PROGRAM MotionControl
VAR
END_VAR

SingleAxis_LD();

METHOD SingleAxis_LD : BOOL
VAR_INPUT
END_VAR
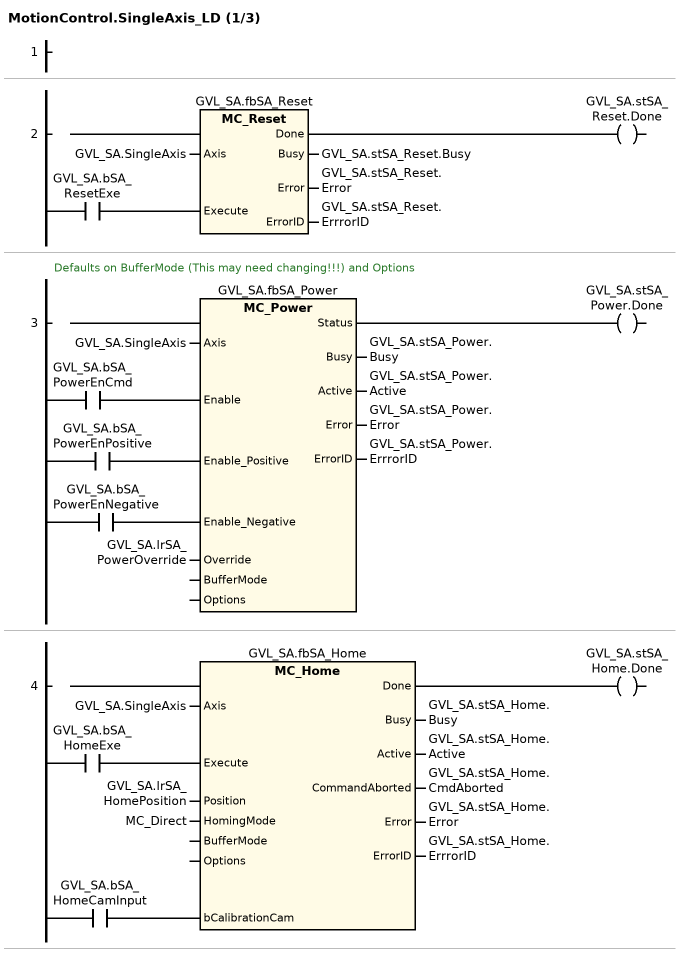
// NETWORK 1

// NETWORK 2
GVL_SA.fbSA_Reset(
    Axis := GVL_SA.SingleAxis,
    Execute := GVL_SA.bSA_ResetExe,
    Busy => GVL_SA.stSA_Reset.Busy,
    Error => GVL_SA.stSA_Reset.Error,
    ErrorID => GVL_SA.stSA_Reset.ErrrorID); // MC_Reset
GVL_SA.stSA_Reset.Done := GVL_SA.fbSA_Reset.Done;

// NETWORK 3
// Defaults on BufferMode (This may need changing!!!) and Options
GVL_SA.fbSA_Power(
    Axis := GVL_SA.SingleAxis,
    Enable := GVL_SA.bSA_PowerEnCmd,
    Enable_Positive := GVL_SA.bSA_PowerEnPositive,
    Enable_Negative := GVL_SA.bSA_PowerEnNegative,
    Override := GVL_SA.lrSA_PowerOverride,
    Busy => GVL_SA.stSA_Power.Busy,
    Active => GVL_SA.stSA_Power.Active,
    Error => GVL_SA.stSA_Power.Error,
    ErrorID => GVL_SA.stSA_Power.ErrrorID); // MC_Power
GVL_SA.stSA_Power.Done := GVL_SA.fbSA_Power.Status;

// NETWORK 4
GVL_SA.fbSA_Home(
    Axis := GVL_SA.SingleAxis,
    Execute := GVL_SA.bSA_HomeExe,
    Position := GVL_SA.lrSA_HomePosition,
    HomingMode := MC_Direct,
    bCalibrationCam := GVL_SA.bSA_HomeCamInput,
    Busy => GVL_SA.stSA_Home.Busy,
    Active => GVL_SA.stSA_Home.Active,
    CommandAborted => GVL_SA.stSA_Home.CmdAborted,
    Error => GVL_SA.stSA_Home.Error,
    ErrorID => GVL_SA.stSA_Home.ErrrorID); // MC_Home
GVL_SA.stSA_Home.Done := GVL_SA.fbSA_Home.Done;

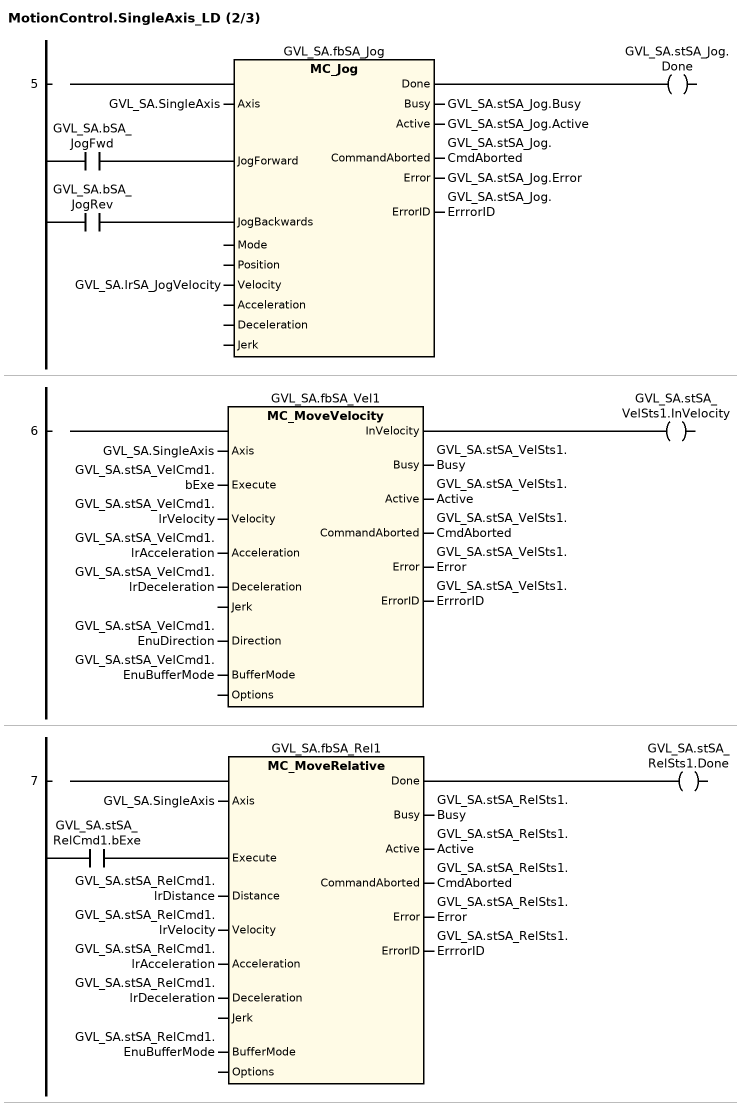
// NETWORK 5
GVL_SA.fbSA_Jog(
    Axis := GVL_SA.SingleAxis,
    JogForward := GVL_SA.bSA_JogFwd,
    JogBackwards := GVL_SA.bSA_JogRev,
    Velocity := GVL_SA.lrSA_JogVelocity,
    Busy => GVL_SA.stSA_Jog.Busy,
    Active => GVL_SA.stSA_Jog.Active,
    CommandAborted => GVL_SA.stSA_Jog.CmdAborted,
    Error => GVL_SA.stSA_Jog.Error,
    ErrorID => GVL_SA.stSA_Jog.ErrrorID); // MC_Jog
GVL_SA.stSA_Jog.Done := GVL_SA.fbSA_Jog.Done;

// NETWORK 6
GVL_SA.fbSA_Vel1(
    Axis := GVL_SA.SingleAxis,
    Execute := GVL_SA.stSA_VelCmd1.bExe,
    Velocity := GVL_SA.stSA_VelCmd1.lrVelocity,
    Acceleration := GVL_SA.stSA_VelCmd1.lrAcceleration,
    Deceleration := GVL_SA.stSA_VelCmd1.lrDeceleration,
    Direction := GVL_SA.stSA_VelCmd1.EnuDirection,
    BufferMode := GVL_SA.stSA_VelCmd1.EnuBufferMode,
    Busy => GVL_SA.stSA_VelSts1.Busy,
    Active => GVL_SA.stSA_VelSts1.Active,
    CommandAborted => GVL_SA.stSA_VelSts1.CmdAborted,
    Error => GVL_SA.stSA_VelSts1.Error,
    ErrorID => GVL_SA.stSA_VelSts1.ErrrorID); // MC_MoveVelocity
GVL_SA.stSA_VelSts1.InVelocity := GVL_SA.fbSA_Vel1.InVelocity;

// NETWORK 7
GVL_SA.fbSA_Rel1(
    Axis := GVL_SA.SingleAxis,
    Execute := GVL_SA.stSA_RelCmd1.bExe,
    Distance := GVL_SA.stSA_RelCmd1.lrDistance,
    Velocity := GVL_SA.stSA_RelCmd1.lrVelocity,
    Acceleration := GVL_SA.stSA_RelCmd1.lrAcceleration,
    Deceleration := GVL_SA.stSA_RelCmd1.lrDeceleration,
    BufferMode := GVL_SA.stSA_RelCmd1.EnuBufferMode,
    Busy => GVL_SA.stSA_RelSts1.Busy,
    Active => GVL_SA.stSA_RelSts1.Active,
    CommandAborted => GVL_SA.stSA_RelSts1.CmdAborted,
    Error => GVL_SA.stSA_RelSts1.Error,
    ErrorID => GVL_SA.stSA_RelSts1.ErrrorID); // MC_MoveRelative
GVL_SA.stSA_RelSts1.Done := GVL_SA.fbSA_Rel1.Done;

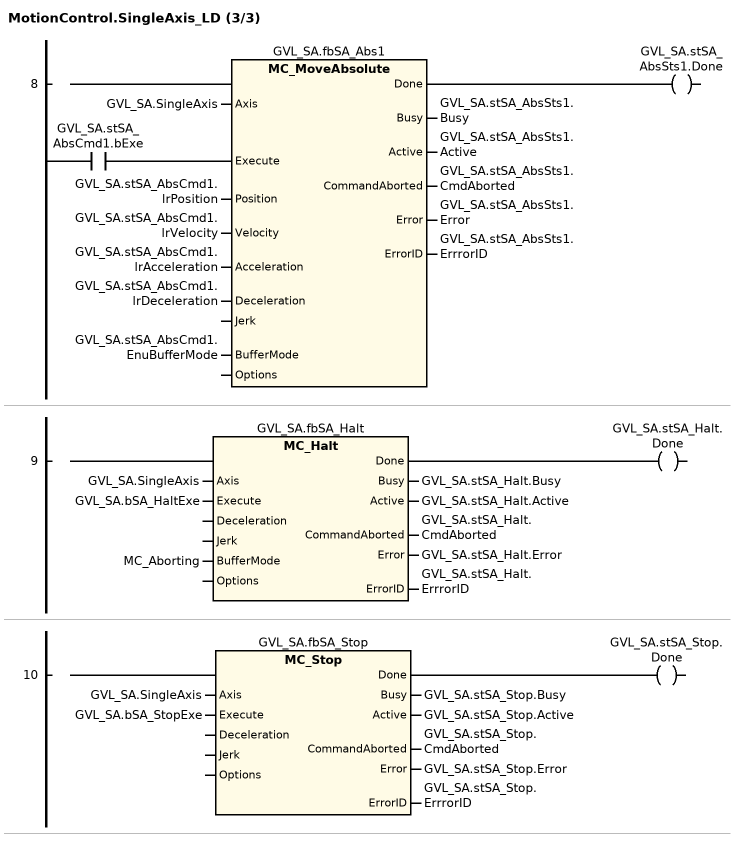
// NETWORK 8
GVL_SA.fbSA_Abs1(
    Axis := GVL_SA.SingleAxis,
    Execute := GVL_SA.stSA_AbsCmd1.bExe,
    Position := GVL_SA.stSA_AbsCmd1.lrPosition,
    Velocity := GVL_SA.stSA_AbsCmd1.lrVelocity,
    Acceleration := GVL_SA.stSA_AbsCmd1.lrAcceleration,
    Deceleration := GVL_SA.stSA_AbsCmd1.lrDeceleration,
    BufferMode := GVL_SA.stSA_AbsCmd1.EnuBufferMode,
    Busy => GVL_SA.stSA_AbsSts1.Busy,
    Active => GVL_SA.stSA_AbsSts1.Active,
    CommandAborted => GVL_SA.stSA_AbsSts1.CmdAborted,
    Error => GVL_SA.stSA_AbsSts1.Error,
    ErrorID => GVL_SA.stSA_AbsSts1.ErrrorID); // MC_MoveAbsolute
GVL_SA.stSA_AbsSts1.Done := GVL_SA.fbSA_Abs1.Done;

// NETWORK 9
GVL_SA.fbSA_Halt(
    Axis := GVL_SA.SingleAxis,
    Execute := GVL_SA.bSA_HaltExe,
    BufferMode := MC_Aborting,
    Busy => GVL_SA.stSA_Halt.Busy,
    Active => GVL_SA.stSA_Halt.Active,
    CommandAborted => GVL_SA.stSA_Halt.CmdAborted,
    Error => GVL_SA.stSA_Halt.Error,
    ErrorID => GVL_SA.stSA_Halt.ErrrorID); // MC_Halt
GVL_SA.stSA_Halt.Done := GVL_SA.fbSA_Halt.Done;

// NETWORK 10
GVL_SA.fbSA_Stop(
    Axis := GVL_SA.SingleAxis,
    Execute := GVL_SA.bSA_StopExe,
    Busy => GVL_SA.stSA_Stop.Busy,
    Active => GVL_SA.stSA_Stop.Active,
    CommandAborted => GVL_SA.stSA_Stop.CmdAborted,
    Error => GVL_SA.stSA_Stop.Error,
    ErrorID => GVL_SA.stSA_Stop.ErrrorID); // MC_Stop
GVL_SA.stSA_Stop.Done := GVL_SA.fbSA_Stop.Done;
END_METHOD

END_PROGRAM

(* stored: Version 1.1.0.1, ProductVersion 3.1.4024.11
   POU MotionControl: Id {5a2c01b0-a377-465c-a2a9-bebb5cce7e25}, SpecialFunc None
   Method SingleAxis_LD: Id {3b3d9a1e-d63e-4a07-bff0-d97af3ca9de8} *)
